# EPICS autosave request: softGlueApp/Db/acquireDma_settings.req
$(P)$(Q)acquireDma.A
$(P)$(Q)acquireDma.B
$(P)$(Q)acquireTranWords
$(P)$(Q)acquireDma.C
$(P)$(Q)acquireDma.SCAN
$(P)$(Q)acquireDma.E
$(P)$(Q)acquireDma.F
$(P)$(Q)acquireDma.H
$(P)$(Q)acquireDmaMode
$(P)$(Q)acquireDma.I
$(P)$(Q)acquireDma.J
$(P)$(Q)acquireDma.K
$(P)$(Q)acquireDma.L
$(P)$(Q)acquireDma.M
$(P)$(Q)acquireDma.N
$(P)$(Q)acquireDma.O
$(P)$(Q)acquireDma.P

$(P)$(Q)acquireDma.PREC

$(P)$(Q)s1name
$(P)$(Q)s2name
$(P)$(Q)s3name
$(P)$(Q)s4name
$(P)$(Q)s5name
$(P)$(Q)s6name
$(P)$(Q)s7name
$(P)$(Q)s8name
